FUNCTION_BLOCK ValveBase_HMI (* Service Interface Function Block Type *)
  (* Standard: 61499-2 *)
  (* Version 1.0.1, 10/17/2023, ApplicationLibDevTeam, Schneider Electric, First Version *)
  PACKAGE Main;
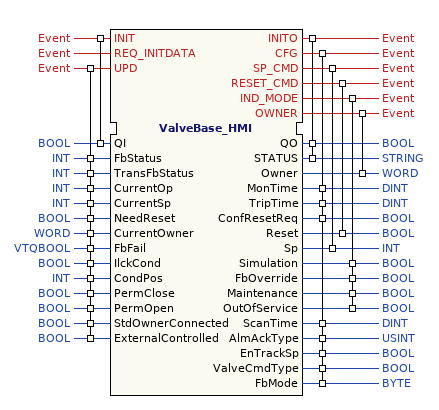
  EVENT_INPUT
    INIT WITH QI;
    REQ_INITDATA; (* Request to initialize data *)
    UPD WITH FbStatus, TransFbStatus, CurrentOp, CurrentSp, NeedReset, CurrentOwner, FbFail, IlckCond, CondPos, PermClose, PermOpen, StdOwnerConnected, ExternalControlled; (* Update data to supervision *)
  END_EVENT
  EVENT_OUTPUT
    INITO WITH QO, STATUS;
    CFG WITH MonTime, TripTime, ConfResetReq, ScanTime, AlmAckType, EnTrackSp, ValveCmdType, FbMode; (* Request for new parameter *)
    SP_CMD WITH Sp; (* Request fro new operator setpoint *)
    RESET_CMD WITH Reset; (* Request  to reset device *)
    IND_MODE WITH Simulation, FbOverride, Maintenance, OutOfService; (* Request for new operational modes *)
    OWNER WITH Owner; (* Request for New Owner *)
  END_EVENT
  VAR_INPUT
    QI : BOOL;
    FbStatus : INT; (* Valve state( 0 = Closed, 1= Opened, 2 = Closed , 253 = Unknown) *) {SET_ATTRIBUTE(Runtime.Archive.Counters, AbsoluteValues=False)} {SET_ATTRIBUTE(Runtime.Archive.Id, 0)} {SET_ATTRIBUTE(Runtime.History.Depth, 100)} {SET_ATTRIBUTE(Runtime.History.SmoothTime, 60000)} {SET_ATTRIBUTE(Runtime.History.SmoothValue, 1)}
    TransFbStatus : INT; (* Valve transition state( 0 = Closed, 1= Opened, 2 = Closed , 6 = Opening, 7= Closing and 253 = Unknown) *) {SET_ATTRIBUTE(Runtime.Archive.Counters, AbsoluteValues=False)} {SET_ATTRIBUTE(Runtime.Archive.Id, 0)} {SET_ATTRIBUTE(Runtime.History.Depth, 100)} {SET_ATTRIBUTE(Runtime.History.SmoothTime, 60000)} {SET_ATTRIBUTE(Runtime.History.SmoothValue, 1)}
    CurrentOp : INT; (* Current value of the output *) {SET_ATTRIBUTE(Runtime.Archive.Counters, AbsoluteValues=False)} {SET_ATTRIBUTE(Runtime.Archive.Id, 1)} {SET_ATTRIBUTE(Runtime.History.Depth, 100)} {SET_ATTRIBUTE(Runtime.History.SmoothTime, 60000)} {SET_ATTRIBUTE(Runtime.History.SmoothValue, 1)}
    CurrentSp : INT; (* Current value of the setpoint *) {SET_ATTRIBUTE(Runtime.Archive.Counters, AbsoluteValues=False)} {SET_ATTRIBUTE(Runtime.Archive.Id, 1)} {SET_ATTRIBUTE(Runtime.History.Depth, 100)} {SET_ATTRIBUTE(Runtime.History.SmoothTime, 60000)} {SET_ATTRIBUTE(Runtime.History.SmoothValue, 1)}
    NeedReset : BOOL; (* 1= Device need reset *)
    CurrentOwner : WORD; (* Current Owner status *)
    FbFail : VTQBOOL; (* 1=Feedback fail alarm status active *)
    IlckCond : BOOL; (* 1= Interlock Active *)
    CondPos : INT; (* Interlock setpoint, 1 = Open , 2 = Close *)
    PermClose : BOOL; (* 1= Close Permission available *)
    PermOpen : BOOL; (* 1= Open Permission available *)
    StdOwnerConnected : BOOL; (* 1 = External owner conncted *)
    ExternalControlled : BOOL; (* 1 = External control is active *)
  END_VAR
  VAR_OUTPUT
    QO : BOOL; (* Event Output Qualifier *)
    STATUS : STRING; (* Service Status *)
    Owner : WORD; (* 16#10= Operator owner , 16#8 = Program owner *)
    MonTime : DINT; (* Feedback monitoring time *)
    TripTime : DINT; (* Feedback trip time *)
    ConfResetReq : BOOL; (* 1= Need reset on confirmation mismatch *)
    Reset : BOOL; (* 1 = Reset request from supervision *)
    Sp : INT; (* New setpoint from the supervision *)
    Simulation : BOOL; (* 1 = Enable device in Simulation *)
    FbOverride : BOOL; (* 1 = Enable device in Override mode *)
    Maintenance : BOOL; (* 1 = Enable device in maintenance mode *)
    OutOfService : BOOL; (* 1 = Out of Service Mode selected *)
    ScanTime : DINT; (* Alarm holding time *)
    AlmAckType : USINT; (* 0=Not ackable; 1=Ack deletes; 2=Came has to be acked; 3=Came and gone have to be acked; 4=Pair has to be acked *)
    EnTrackSp : BOOL; (* 1= Enable the tracking of Interlock setpoint *)
    ValveCmdType : BOOL; (* 0 = Normally Closed Valve, 1 = Normally Open Valve *)
    FbMode : BYTE; (* Bit mask to disable feedback monitoring (16#0- Both fb; 16#1- Only Open fb; 16#3- No fb) *)
  END_VAR
  SERVICE /
    SEQUENCE 
    END_SEQUENCE
  END_SERVICE
END_FUNCTION_BLOCK
